# B&R Automation Studio project JOB_NUMBER (part 6)

#### SafetyUI.var - Local variables
```iecst
(********************************************************************
 * COPYRIGHT -- Bernecker + Rainer
 ********************************************************************
 * Program: SafetySample
 * File: SafetySample.var
 * Author: B&R
 ********************************************************************
 * Local variables of program SafetySample
 ********************************************************************)
VAR
	appcmd1 : DownloadCmdApplicationTypeV1; (*command structure for application download*)
	dataAcknMachineOptions : DownloadAcknMaOpTypeV1; (*data to acknowledge bit machine options*)
	datacmd1 : DownloadCmdMaOpTypeV1; (*command structure for machine options download*)
	datacmd2 : DownloadCmdExtMaOpTypeV1; (*command structure for extended machine options download*)
	dataMachineOptionsBitInput : ConfigurationBitOptionsTypeV1; (*data for bit machine options*)
	dataModuleFlagsInput : ConfigurationModuleFlagsTypeV1; (*data for module flags*)
	dialogApplication : BOOL; (*visualization dialog for application download*)
	dialogButtonLeft : BOOL; (*left button in visualization dialog*)
	dialogButtonRight : BOOL; (*right button in visualization dialog*)
	dialogData : BOOL; (*visualization dialog for machine options download*)
	dialogExtData : BOOL; (*visualization dialog for extended machine options download*)
	dialogRemoteCmd : BOOL; (*visualization dialog for remote control*)
	executeapp1 : BOOL; (*execute application download*)
	executedata1 : BOOL; (*execute machine options download*)
	executedata2 : BOOL; (*execute extended machine options download*)
	executeRemoteCmd : BOOL; (*execute remote control*)
	indexButtonLeft : UINT; (*index for button text*)
	indexButtonRight : UINT; (* index for button text*)
	indexCompareTextData : UINT; (*index for compare message machine options*)
	indexCompareTextExtData : UINT; (*index for compare message extended machine options*)
	indexFAILLed : UINT; (*index FAIL led*)
	indexFwAcknLed : UINT; (*index FW-ACKN led*)
	indexHeaderText : UINT; (*index dialog header text*)
	indexMessageText : UINT; (*index message text*)
	indexMxchgLed : UINT; (*index MXCHG led*)
	indexRELed : UINT; (*index R/E led*)
	Interface : STRING[80] := ''; (*interface information for SafeLOGIC*)
	Node : USINT; (*node information for SafeLOGIC*)
	pDeviceListOut : REFERENCE TO ARRAY[0..1] OF ConfigurationDeviceTypeV1; (*device list from FUB*)
	pMachineOptionsBitOut : REFERENCE TO ConfigurationBitOptionsTypeV1; (*bit machine options from FUB*)
	pModuleFlagsOut : REFERENCE TO ConfigurationModuleFlagsTypeV1; (*module flags form FUB*)
	readUDIDhighSL : EplSDORead; (*function block to read UDID high from device*)
	readUDIDhighSLX : AsIOAccRead; (*function block to read UDID high from device*)
	readUDIDlowSL : EplSDORead; (*function block to read UDID low from device*)
	readUDIDlowSLX : AsIOAccRead; (*function block to read UDID low from device*)
	remotecmd : RemoteControlCmdTypeV1; (*command structure for remote control*)
	safeDownloadApplication_0 : safeDownloadApplication; (*function block safeDownloadApplication*)
	safeDownloadData_0 : safeDownloadData; (*function block safeDownloadData*)
	safeDownloadData_1 : safeDownloadData; (*function block safeDownloadData*)
	safeRemoteControl_0 : safeRemoteControl; (*function block safeRemoteControl*)
	slxused : BOOL; (*SafeLOGIC-X is used*)
	Station : STRING[80] := 'IF6.ST1'; (*station information for SafeLOGIC-X*)
	statusAcknInfoData : UINT; (*acknowledge boxes for machine options*)
	statusAcknInfoExtData : UINT; (*acknowledge boxes for extended machine options*)
	statusButtonActiv : ARRAY[0..15] OF USINT; (*button activ*)
	statusButtonInactiv : ARRAY[0..15] OF USINT; (*button inactiv*)
	statusButtonUnlockApp : UINT; (*unlock buttons application*)
	statusButtonUnlockData : UINT; (*unlock buttons data*)
	statusButtonUnlockExtData : UINT; (*unlock buttons extended data*)
	statusDialog : UINT; (*dialog box*)
	statusSetPassword : UINT; (*visualization status to set password*)
	statusSLInformation : UINT; (*display information for SafeLOGIC*)
	stautsSLXInformation : UINT; (*display information for SafeLOGIC-X*)
	UDID_High : UINT; (*UDID_high for SafelOGIC*)
	UDID_Low : UDINT; (*UDID_low for SafeLOGIC*)
	visuAcknExtData : DownloadAcknExtMaOpTypeV1; (*acknowledge extended machine options*)
	visuAcknMachineOptions : ARRAY[0..511] OF BOOL; (*acknowledge machine options*)
	visuApplicationCRC : STRING[8]; (*CRC HEX string for visualization*)
	visuDeviceListInput : ARRAY[0..1] OF DownloadDeviceTypeV1; (*device list input*)
	visuDeviceListOutput : ARRAY[0..1] OF DownloadDeviceTypeV1; (*device list output*)
	visuDintInput : ConfigurationDintOptionsTypeV1; (*DINT channels input*)
	visuDintOutput : ConfigurationDintOptionsTypeV1; (*DINT channels output*)
	visuEnableDINTOptions : BOOL; (*enable DINT options*)
	visuEnableINTOptions : BOOL; (*enable INT options*)
	visuEnableMachineOptions : BOOL; (*enable BIT options*)
	visuEnableModuleFlags : BOOL; (*enable module flags*)
	visuEnableUDINTOptions : BOOL; (*enable UDINT options*)
	visuEnableUINTOptions : BOOL; (*enable UINT options*)
	visuIntInput : ConfigurationIntOptionsTypeV1; (*INT channels input*)
	visuIntOutput : ConfigurationIntOptionsTypeV1; (*INT channels output*)
	visuMachineOptionsBitInput : ARRAY[0..511] OF BOOL; (*BIT options input*)
	visuMachineOptionsBitOutput : ARRAY[0..511] OF BOOL; (*BIT options output*)
	visuModuleFlagsNotPresentInput : ARRAY[0..1023] OF BOOL; (*not present module flags input*)
	visuModuleFlagsNotPresentOutput : ARRAY[0..1023] OF BOOL; (*not present module flags output*)
	visuModuleFlagsOptionalInput : ARRAY[0..1023] OF BOOL; (*optional module flags input*)
	visuModuleFlagsOptionalOutput : ARRAY[0..1023] OF BOOL; (*optional module flags output*)
	visuModuleFlagsStartupInput : ARRAY[0..1023] OF BOOL; (*startup module flags input*)
	visuModuleFlagsStartupOutput : ARRAY[0..1023] OF BOOL; (*startup module flags output*)
	visuUDID_High : STRING[8]; (*UDID hex string for visualization*)
	visuUDID_Low : STRING[8]; (*UDID hex string for visualization*)
	visuUdintInput : ConfigurationUdintOptionsTypeV1; (*UDINT channels input*)
	visuUdintOutput : ConfigurationUdintOptionsTypeV1; (*UDINT channels output*)
	visuUintInput : ConfigurationUintOptionsTypeV1; (*UINT channels input*)
	visuUintOutput : ConfigurationUintOptionsTypeV1; (*UINT channels output*)
	visuUsedSLIDData : UINT; (*SafeLOGIC ID for data download*)
	visuUsedSLIDRemote : UINT; (*SafeLOGIC ID for remote control*)
	xcnt : UINT; (*counter variable*)
	strStatusID : STRING[10];
	strMXCHG_Led : STRING[10];
	strFWACKN_Led : STRING[10];
	strStatus : STRING[10];
	strRE_Led : STRING[10];
	strFAIL_Led : STRING[10];
	strMessageTest : STRING[10];
	bVisAppButtons : BOOL;
	bVisInterfaceNode : BOOL;
	bVisStation : BOOL;
	strDownloadStatus : STRING[10];
	strDataStatus : STRING[10];
	strSKFormatStyle : STRING[15];
	strSKXCHGtStyle : STRING[15];
	strScanStyle : STRING[15];
	strAck1Style : STRING[15];
	strAck2Style : STRING[15];
	strAck3Style : STRING[15];
	strAck4Style : STRING[15];
	strAckNStyle : STRING[15];
	strFWACKNStyle : STRING[15];
	strTestStyle : STRING[15];
	strClearStyle : STRING[15];
	safeLogicStatus : RemoteControlStatusTypeV1;
	visuEnableButtons : BOOL;
	safety : USINT;
	execute : BOOL;
	remoteControlcmd : REFERENCE TO RemoteControlCmdTypeV1;
	executeRemoteControl : BOOL;
	remoteCmdGetStatus : RemoteControlCmdTypeV1;
	ton_refreshStatus : TON_10ms;
	safePLC_Ok : BOOL;
	getNode : getNodeFromPV;
END_VAR
```

### Package Logical/COMMUNICATION - COMMUNICATION

### Communication.var
```iecst
(*Comm Config*)
VAR CONSTANT
  UDP_COMM_PORT : UINT := 4004;
  TCP_COMM_PORT : UINT := 12005;
END_VAR
(*Data sizes*)
VAR CONSTANT
  EVUE_COMM_BUFFER_SIZE : UINT := 16000; (*Size of data array for the memory map*)
  TCP_SEND_BUFFER_SIZE : UINT := 1000; (**Size of the send buffer for responses*)
  TCP_RECV_BUFFER_SIZE : UINT := 16000; (**Size of the recieve buffer*)
  UDP_SEND_PACKET_SIZE : UINT := 4000; (**Size of the packet to send*)
END_VAR
(***********UDP Comm Config************)
VAR CONSTANT
  LIVE_DATA_MAX_CONNECTIONS : USINT := 5; (**Maximum number of UDP Connections*)
  LIVE_DATA_MAX_POOL_SIZE : USINT := 10; (**Maximum number of data transmissions on 1 connection*)
END_VAR
(**)
(*DATA TYPE DEFINITIONS*)
VAR CONSTANT
  LIVE_DATA_TYPE_EVUE_UDP_COMM_1 : UINT := 1;
  LIVE_DATA_TYPE_EVUE_UDP_COMM_2 : UINT := 2;
  LIVE_DATA_TYPE_EVUE_UDP_COMM_3 : UINT := 3;
  LIVE_DATA_TYPE_EVUE_UDP_COMM_4 : UINT := 4;
  LIVE_DATA_TYPE_RAIL_MESSAGES : UINT := 1001;
END_VAR
(*DATA TYPE DEFINITIONS*)
VAR
        CommArray : ARRAY[0..EVUE_COMM_BUFFER_SIZE] OF UDINT; (**Global Array of pointers of comm vars*)
END_VAR
```

### Library Logical/COMMUNICATION/MbusTCP (ANSIC, version 1.39.0)
Depends on: astcp, asstring, standard, AsARCfg, sys_lib

### Program Logical/COMMUNICATION/ModSlave (IEC, version 2.00.1) - ModSlave

#### ModSlave.st - Init, cyclic, exit code
```iecst
(********************************************************************
  * COPYRIGHT --
  ********************************************************************
  * PROGRAM: ModSlave
  ********************************************************************
  * Implementation OF PROGRAM ModSlave
  ********************************************************************)

PROGRAM _INIT
  (* --------------------------------------------------------------------
    Reset FUNCTION blocks AND data structure on startup (SGC)
    --------------------------------------------------------------------- *)
  memset(ADR(ModbusTcpSlave), 0, SIZEOF(ModbusTcpSlave));
  memset(ADR(SlaveConfig), 0, SIZEOF(SlaveConfig));
  memset(ADR(logger), 0, SIZEOF(logger));

  (* --------------------------------------------------------------------
    Create default IO mapping FOR digital AND analog area
    --------------------------------------------------------------------- *)

  FOR idx:=0 TO SIZEOF(EVUE_MODBUS)/SIZEOF(EVUE_MODBUS[0])-1 DO
    SlaveConfig.p_holding_registers[idx] := ADR(EVUE_MODBUS[idx]);
  END_FOR;

  (* --------------------------------------------------------------------
    Configure FUNCTION block instance
    --------------------------------------------------------------------- *)
  ModbusTcpSlave.enable			:= 1; 					(* Enable function block *)
  ModbusTcpSlave.device			:= ADR('IF3');			(* Ethernet device string *)
  ModbusTcpSlave.p_cfg			:= ADR(SlaveConfig); 	(* IO configuration *)
  ModbusTcpSlave.master_timeout 	:= 5000; 			     	(* Disconnect master after x miliseconds when no request was sent, 0 = disabled *)

  (* The LOG information will show communication details. Enable for debugging,
  disable FOR production TO save system resources *)

  ModbusTcpSlave.log.data_lines 	:= 20; 					(* Number of logging lines *)
  ModbusTcpSlave.log.pData 		:= ADR(logger);			(* Pointer to logger string array *)
  mbSlaveStep := 1;
END_PROGRAM

PROGRAM _CYCLIC

  CASE mbSlaveStep OF
    0:
      (* --------------------------------------------------------------------
        Reset FUNCTION blocks AND data structure on startup (SGC)
        --------------------------------------------------------------------- *)
      memset(ADR(ModbusTcpSlave), 0, SIZEOF(ModbusTcpSlave));
      memset(ADR(SlaveConfig), 0, SIZEOF(SlaveConfig));
      memset(ADR(logger), 0, SIZEOF(logger));

      (* --------------------------------------------------------------------
        Configure FUNCTION block instance
        --------------------------------------------------------------------- *)
      ModbusTcpSlave.enable			:= 1; 					(* Enable function block *)
      ModbusTcpSlave.device			:= ADR('IF3');			(* Ethernet device string *)
      ModbusTcpSlave.p_cfg			:= ADR(SlaveConfig); 	(* IO configuration *)
      ModbusTcpSlave.master_timeout 	:= 5000; 			     	(* Disconnect master after x miliseconds when no request was sent, 0 = disabled *)

      // Go to mbSlaveStep 1
      mbSlaveStep := 1;

    1:
      // Call MbSlave FUB
      ModbusTcpSlave();
  END_CASE

  (* --------------------------------------------------------------------
    Reset last error information
    --------------------------------------------------------------------- *)
  IF(reset_error) THEN
    memset(ADR(ModbusTcpSlave.last_error), 0, 2);
    reset_error := 0;
  END_IF
END_PROGRAM
```

### Program Logical/COMMUNICATION/udpComm (IEC, version 2.00.1) - udpComm

#### Main.st - Init, cyclic, exit code
```iecst
(*
  ----------------------------------------------------------------------------------------------------------------------------------------
  --LIVE DATA TASK--
  UDP MAX FRAME SIZE IS 65507 Bytes
  -----------------------------------------------------------------------------------------------------------------------------------------
  *)
  //V1.00.1 -- 06/09/2019 -- First Version
  //V1.00.2 -- 05/01/2020 -- Clean up basic version + Add dynamic start up for ABB drive data
  //V2.00.1 -- 11/03/2020 -- Add Structures to replace TCP/IP Driver
  PROGRAM _INIT
  //Configure a static connection (Testing)
  LiveDataConnection[1].Config.ServerIP 		:= eVueServerIP;
  LiveDataConnection[1].Config.ServerPort		:= UDP_COMM_PORT;
  LiveDataConnection[1].Config.Type 			:= LIVE_DATA_CONFIG_STATIC;
  //Create a fix request pool for test
  LiveDataConnection[1].RequestPool.PoolList[1] 	:= LIVE_DATA_TYPE_EVUE_UDP_COMM_1;
  LiveDataConnection[1].RequestPool.PoolList[2] 	:= LIVE_DATA_TYPE_EVUE_UDP_COMM_2;
  LiveDataConnection[1].RequestPool.PoolList[3] 	:= LIVE_DATA_TYPE_EVUE_UDP_COMM_3;
  LiveDataConnection[1].RequestPool.PoolList[4] 	:= LIVE_DATA_TYPE_EVUE_UDP_COMM_4;
  LiveDataConnection[1].RequestPool.PoolList[5] 	:= LIVE_DATA_TYPE_RAIL_MESSAGES;
  LiveDataConnection[1].RequestPool.PoolListSize 	:= 5;
  _initialiseComms;
  END_PROGRAM

  PROGRAM _CYCLIC

    IF EDGEPOS(udpIdent_Error) THEN
      udpCloseAllIdent := 0;
      n := 0;
    END_IF;
    IF udpIdent_Error THEN // We have too many ports open -- temp stop all clients and close all udp connections.

      CASE udpCloseAllIdent OF

      0://Get list off all open idents
        ioctl ACCESS ADR(udpIoctl_Error);
        ioctl.enable := 1;
        ioctl.ident := udpINVALID_IDENT;
        ioctl.ioctl := udpID_LIST_GET;
        ioctl.pData := ADR(identInfo.IdentsList[0]);
        ioctl.datalen := SIZEOF(identInfo.IdentsList);
        ioctl();
        IF (ioctl.status = ERR_OK) THEN
          udpCloseAllIdent := 1;
        ELSIF (ioctl.status <> ERR_FUB_BUSY) THEN

        END_IF;

      1://Close all open connections

        close ACCESS ADR(udpClose_Error);
        close.enable := (identInfo.IdentsList[n] > 0);
        close.ident := identInfo.IdentsList[n];
        close();
        IF (close.status = ERR_OK) OR ((close.status <> ERR_FUB_BUSY) AND (close.status <> ERR_FUB_ENABLE_FALSE)) THEN
          identInfo.IdentsList[n] := 0;
          IF (n < 199) THEN
            n := n + 1;
          ELSE
            udpCloseAllIdent := 2;
          END_IF;
        ELSIF (identInfo.IdentsList[n] = 0) THEN
          udpCloseAllIdent := 2;
        END_IF;

      2:// Reinint all connections
        FOR n := 1 TO LIVE_DATA_MAX_CONNECTIONS DO
          connection ACCESS ADR(LiveDataConnection[n]);
          connection.State := LIVE_DATA_INIT;
        END_FOR;
        udpIdent_Error := 0;
        udpCloseAllIdent := 0;
      END_CASE;

    ELSE //Run
      FOR n := 1 TO LIVE_DATA_MAX_CONNECTIONS DO
        connection ACCESS ADR(LiveDataConnection[n]);
        CASE connection.State  OF
          LIVE_DATA_INIT: //Every connection must be initialised with server IP and Port. This can be static or dynamic via http GET.
            CASE connection.Config.Type OF
              LIVE_DATA_CONFIG_STATIC:
                //Check the IP is valid
                IF connection.Config.ServerIP <> '' THEN //Don;t check Port as this could be 0
                  connection.State := LIVE_DATA_WAIT;
                END_IF;
              LIVE_DATA_CONFIG_DYNAMIC_CLIENT:
                //Http request to load the Server details + current request pool
              LIVE_DATA_CONFIG_DYNAMIC_SERVER;
                //Wait for a request on the http server to start a connection.
            END_CASE;

          LIVE_DATA_WAIT:
            _AddRemoveFromPool;
            //Wait for the Request pool to be greater than 0
            IF (connection.RequestPool.PoolListSize > 0) THEN
              connection.State := LIVE_DATA_OPEN_CONNECTION;
            END_IF;

          LIVE_DATA_OPEN_CONNECTION:
            //Open connection to serverr
            open ACCESS ADR(connection.Functions.Open);
            open.enable 	:= 1;
            open.options	:= 0;
            open.pIfAddr 	:= 0;//
            open.port		:= 0;//
            open();
            IF (open.status = ERR_OK) THEN
              connection.State := LIVE_DATA_SETUP_CONNECTION_TOS;
            ELSIF (open.status <> ERR_FUB_BUSY) THEN
              connection.Error := open.status;
              connection.State := LIVE_DATA_ERROR; // Go directly to error as the connection has failed
            END_IF;

          LIVE_DATA_SETUP_CONNECTION_TOS://Configure the UDP
            //We must set
            //1) Type of service 	-- udpIP_TOS_SET -- udpIP_TOS_RELIABILITY
            //2) Time to live 		--
            //Optional Send Buffer	-- udpSO_SNDBUF_SET

            //				udpIP_TOS_LOWDELAY			16
            //				udpIP_TOS_THROUGHPUT		8
            //				udpIP_TOS_RELIABILITY		4
            //				udpIP_TOS_MINCOST			2

            ioctl ACCESS ADR(connection.Functions.Ioctl);
            ioctl.enable := 1;
            ioctl.ident := connection.Functions.Open.ident;
            ioctl.ioctl := udpIP_TOS_SET;
            ioctl.pData := ADR(connection.Config.TOS);
            ioctl.datalen := 4;
            ioctl();
            IF (ioctl.status = ERR_OK) THEN
              connection.State := LIVE_DATA_SETUP_CONNECTION_TTL;
            ELSIF (ioctl.status <> ERR_FUB_BUSY) THEN
              connection.Error := ioctl.status;
              connection.State := LIVE_DATA_CLOSE_CONNECTION;
            END_IF;

          LIVE_DATA_SETUP_CONNECTION_TTL: //Time to LIVE in seconds -- MAX 255

            ioctl ACCESS ADR(connection.Functions.Ioctl);
            ioctl.enable := 1;
            ioctl.ident := connection.Functions.Open.ident;
            ioctl.ioctl := udpIP_TTL_SET;
            ioctl.pData := ADR(connection.Config.TTL);
            ioctl.datalen := 4;
            ioctl();
            IF (ioctl.status = ERR_OK) THEN
              connection.State := LIVE_DATA_CONNECT;
            ELSIF (ioctl.status <> ERR_FUB_BUSY) THEN
              connection.Error := ioctl.status;
              connection.State := LIVE_DATA_CLOSE_CONNECTION;
            END_IF;

          LIVE_DATA_CONNECT: // Connect to a specific Device (this is optional but improves performance)
            connect	ACCESS ADR(connection.Functions.Connect);
            connect.enable 	:= 1;
            connect.ident 	:= connection.Functions.Open.ident;
            connect.pHost	:= ADR(connection.Config.ServerIP);
            connect.port 	:= connection.Config.ServerPort;
            connect();
            IF (connect.status = ERR_OK) THEN
              IF getIdentInfo THEN
                connection.State := LIVE_DATA_GET_IDENT_LIST;
              ELSE
                connection.State := LIVE_DATA_BUILD_DATA;
              END_IF;
            ELSIF (connect.status <> ERR_FUB_BUSY) THEN
              connection.Error := connect.status;
              connection.State := LIVE_DATA_DISCONNECT;
            END_IF;
          LIVE_DATA_BUILD_DATA:
            //Build data-- Build a header and data combined.
            //Byte 1 		-- Request Type USINT
            //Byte 2 & 3	-- Header Size(Bytes) UINT
            //Byte 4,5,6,7	-- CheckSum		UDINT
            //Byte xxx		-- HEADER INFO -- BESPOKE TO Request Type
            //DATA--
            IF (connection.RequestPool.Pointer > 0) THEN
              CASE connection.RequestPool.PoolList[connection.RequestPool.Pointer] OF

                LIVE_DATA_TYPE_EVUE_UDP_COMM_1..LIVE_DATA_TYPE_EVUE_UDP_COMM_4:
                  //Built the packet
                  udpComm[0] := connection.RequestPool.Pointer;
                  FOR n := 1 TO UDP_SEND_PACKET_SIZE DO
                    pointer :=  n + (UDP_SEND_PACKET_SIZE * (udpComm[0] - 1));
                    IF (CommArray[pointer] <> 0) AND (pointer <= EVUE_COMM_BUFFER_SIZE) THEN
                      brsmemcpy(ADR(udpComm[n]),CommArray[pointer],2);
                    ELSE
                      udpComm[n] := 0;
                    END_IF;
                  END_FOR;
                  pData := ADR(udpComm);
                  length := SIZEOF(udpComm);
                  connection.State := LIVE_DATA_SEND_DATA;

                LIVE_DATA_TYPE_RAIL_MESSAGES:// Rail messages
                  messages[0] := LIVE_DATA_TYPE_RAIL_MESSAGES;
                  FOR n := 1 TO RAIL_COUNT DO
                    messages[n] := RailComm[n].Messages.Write;
                  END_FOR;
                  pData := ADR(messages);
                  length := SIZEOF(messages);
                  connection.State := LIVE_DATA_SEND_DATA;

                ELSE
                  //Invalid type- Check the pool again
                  connection.State := LIVE_DATA_CHECK_REQUESTPOOL;
              END_CASE;
            ELSE
              connection.State := LIVE_DATA_CHECK_REQUESTPOOL;
            END_IF;

          LIVE_DATA_SEND_DATA:
            send ACCESS ADR(connection.Functions.Send);
            send.enable 	:= 1;
            send.ident 		:= connection.Functions.Open.ident;
            send.flags 		:= udpMSG_DONTROUTE;// Do not send via the gateway- Route Directly to Server
            send.pData 		:= pData;
            send.datalen	:= length;
            send();
            IF (send.status = ERR_OK) THEN
              connection.State := LIVE_DATA_CHECK_REQUESTPOOL;
            ELSIF send.status = udpERR_CONNREFUSED THEN // Server is not there, disconnect and start again
              connection.State := LIVE_DATA_DISCONNECT;
            ELSIF (send.status <> ERR_FUB_BUSY) THEN
              connection.Error := send.status;
              connection.State := LIVE_DATA_DISCONNECT;
            END_IF;

            //send.pHost || THESE ARE IGNORED BECAUSE WE ARE MAKING A DIRECT CONNECTION USING THE CONNECT FUB||
            //send.port

          LIVE_DATA_CHECK_REQUESTPOOL:
            //Check that the request pool hasn;t changed- Shuffle to the next Requested packet.
            _AddRemoveFromPool;
            //IF the pool is empty close the connection and wait
            IF (connection.RequestPool.Pointer = 0) AND (connection.RequestPool.PoolListSize > 0) THEN
              connection.RequestPool.Pointer := 1;
            ELSIF (connection.RequestPool.Pointer = connection.RequestPool.PoolListSize) THEN
              connection.RequestPool.Pointer := 1;
            ELSIF (connection.RequestPool.Pointer < connection.RequestPool.PoolListSize) THEN
              connection.RequestPool.Pointer := connection.RequestPool.Pointer + 1;
            ELSIF (connection.RequestPool.Pointer > connection.RequestPool.PoolListSize) AND (connection.RequestPool.PoolListSize > 0) THEN
              connection.RequestPool.Pointer := 1;
            END_IF;

            validConnection := (connection.Config.ServerIP <> '');
            IF (connection.RequestPool.PoolListSize = 0) OR NOT validConnection THEN
              connection.State := LIVE_DATA_DISCONNECT;
            ELSE
              connection.State := LIVE_DATA_BUILD_DATA;
            END_IF;

          LIVE_DATA_DISCONNECT:
            disconnect ACCESS ADR(connection.Functions.Disconnect);
            disconnect.enable := 1;
            disconnect.ident := connection.Functions.Open.ident;
            disconnect();
            IF (disconnect.status = ERR_OK) THEN
              connection.State := LIVE_DATA_CLOSE_CONNECTION;
            ELSIF (disconnect.status <> ERR_FUB_BUSY) THEN
              connection.Error := disconnect.status;
              connection.State := LIVE_DATA_CLOSE_CONNECTION;
            END_IF;

          LIVE_DATA_CLOSE_CONNECTION:
            close ACCESS ADR(connection.Functions.Close);
            close.enable := 1;
            close.ident := connection.Functions.Open.ident;
            close();
            IF (close.status = ERR_OK) THEN
              IF (connection.Error > 0) THEN
                connection.State := LIVE_DATA_ERROR;
              ELSE
                connection.State := LIVE_DATA_INIT;
              END_IF;
              IF (connection.Config.Type <> LIVE_DATA_CONFIG_STATIC) THEN
                connection.RequestPool 			:= CLEAR_REQUEST_POOL;
                connection.Config.ServerIP 		:= '';
                connection.Config.ServerPort 	:= 0;
              END_IF;

            ELSIF (close.status <> ERR_FUB_BUSY) THEN
              connection.Error := close.status ;
              connection.State := LIVE_DATA_ERROR;
            END_IF;

          LIVE_DATA_ERROR:
            IF (connection.Error = udpERR_NOMORE_IDENTS) THEN
              // All Idents are used we have to close them manually.
              udpIdent_Error := 1;
            ELSE
              errorCount := errorCount + 1;
              connection.Error := 0;
              connection.State := LIVE_DATA_INIT;
            END_IF;

          LIVE_DATA_GET_IDENT_LIST:
            ioctl ACCESS ADR(connection.Functions.Ioctl);
            ioctl.enable := 1;
            ioctl.ident := udpINVALID_IDENT;
            ioctl.ioctl := udpID_LIST_GET;
            ioctl.pData := ADR(identInfo.IdentsList[0]);
            ioctl.datalen := SIZEOF(identInfo.IdentsList);
            ioctl();
            IF (ioctl.status = ERR_OK) THEN
              connection.State := LIVE_DATA_GET_IDENT_MAX;
            ELSIF (ioctl.status <> ERR_FUB_BUSY) THEN

            END_IF;

          LIVE_DATA_GET_IDENT_MAX:
            ioctl ACCESS ADR(connection.Functions.Ioctl);
            ioctl.enable := 1;
            ioctl.ident := udpINVALID_IDENT;
            ioctl.ioctl := udpID_MAX_GET;
            ioctl.pData := ADR(identInfo.MaxIdents);
            ioctl.datalen := 4;
            ioctl();
            IF (ioctl.status = ERR_OK) THEN
              connection.State := LIVE_DATA_BUILD_DATA;
            ELSIF (ioctl.status <> ERR_FUB_BUSY) THEN

            END_IF;

        END_CASE;

      END_FOR;
    END_IF;

  END_PROGRAM

  PROGRAM _EXIT
    // DO we have to close the connections on EXIT -- Perhaps when a transfer happens!!

  END_PROGRAM
```

#### _AddRemoveFromPool.st
```iecst
ACTION _AddRemoveFromPool:
IF (connection.RequestPool.AddToPool > 0) THEN
  //Check the requested frame is not already in the list
  FOR i := 1 TO LIVE_DATA_MAX_POOL_SIZE DO
    IF (connection.RequestPool.PoolList[i] = connection.RequestPool.AddToPool) THEN
      connection.RequestPool.AddToPool := 0;
      EXIT;
    ELSIF (connection.RequestPool.PoolList[i] = 0) THEN
      EXIT;
    END_IF;
  END_FOR;

  IF (connection.RequestPool.AddToPool > 0) THEN //Check we haven't already found the request in the pool
    IF (connection.RequestPool.PoolListSize < LIVE_DATA_MAX_POOL_SIZE) THEN //Keep in range
      connection.RequestPool.PoolListSize := connection.RequestPool.PoolListSize + 1;
      connection.RequestPool.PoolList[connection.RequestPool.PoolListSize] := connection.RequestPool.AddToPool;
      connection.RequestPool.AddToPool := 0;
    END_IF;
  END_IF;
END_IF;
IF (connection.RequestPool.RemoveFromPool > 0) THEN
  //Find the pool in the array-- Remove it then shuffle the list.
  FOR i := 1 TO LIVE_DATA_MAX_POOL_SIZE DO
    IF (connection.RequestPool.PoolList[i] = connection.RequestPool.RemoveFromPool) THEN
      //Shuffle the list
      brsmemmove(ADR(connection.RequestPool.PoolList[i]),ADR(connection.RequestPool.PoolList[i + 1]),((LIVE_DATA_MAX_POOL_SIZE - i)*2));
      //connection.RequestPool.PoolList[LIVE_DATA_MAX_POOL_SIZE] := 0;
      connection.RequestPool.PoolListSize := connection.RequestPool.PoolListSize - 1;
      IF (connection.RequestPool.PoolListSize > LIVE_DATA_MAX_POOL_SIZE) THEN
        connection.RequestPool.PoolListSize := 0;
      END_IF;
      EXIT;
    ELSIF (connection.RequestPool.PoolList[i] = 0) THEN
      EXIT; //Not found
    END_IF;
  END_FOR;
  connection.RequestPool.RemoveFromPool := 0;
END_IF;
END_ACTION
```

#### _initialiseComms.st
```iecst
// Initialise the Comm registers.
ACTION _initialiseComms:
  //Generated Init Code.
  FOR n := 0 TO EVUE_COMM_BUFFER_SIZE DO
    CommArray[n] := 0;
  END_FOR;

END_ACTION
```

#### Types.typ - Local data types
```iecst
TYPE
  identInfo_typ : 	STRUCT
    MaxIdents : UDINT;
    IdentsList : ARRAY[0..199]OF UDINT;
  END_STRUCT;
END_TYPE
```

#### Variables.var - Local variables
```iecst
VAR CONSTANT
  CLEAR_REQUEST_POOL : LiveData_RequestPool_typ := (AddToPool:=0,RemoveFromPool:=0,PoolListSize:=0,Pointer:=0);
END_VAR
VAR
  n : UINT;
  pointer : UDINT;
  connection : REFERENCE TO LiveDataConnection_typ;
  LiveDataConnection : ARRAY[1..LIVE_DATA_MAX_CONNECTIONS] OF LiveDataConnection_typ;
  udpComm : ARRAY[0..UDP_SEND_PACKET_SIZE] OF UINT;
  open : REFERENCE TO UdpOpen;
  ioctl : REFERENCE TO UdpIoctl;
  connect : REFERENCE TO UdpConnect;
  send : REFERENCE TO UdpSend;
  pData : UDINT;
  length : UDINT;
  disconnect : REFERENCE TO UdpDisconnect;
  close : REFERENCE TO UdpClose;
  errorCount : UDINT;
  validConnection : BOOL;
  i : USINT;
  identInfo : identInfo_typ;
  getIdentInfo : BOOL;
  udpIdent_Error : BOOL;
  udpIoctl_Error : UdpIoctl;
  udpCloseAllIdent : USINT;
  udpClose_Error : UdpClose;
  data : ARRAY[0..65534] OF SINT; (**Max data frame that can be sent by UDP*)
  messages : ARRAY[0..RAIL_COUNT] OF UINT;
END_VAR
```

### Program Logical/COMMUNICATION/tcpComm (IEC, version 1.00.1) - tcpComm

#### Main.st - Init, cyclic, exit code
```iecst
//V1.00 	- First Version
//V1.00.1 	- ADD Evue modbus decode function.
PROGRAM _INIT
  _initialiseComms;
	listenPort 	:= TCP_COMM_PORT;
	socketState := TCP_SOCKET_OPEN;
END_PROGRAM
PROGRAM _CYCLIC

	CASE socketState OF
		TCP_SOCKET_OPEN:
			tcpOpen.enable := 1;
			tcpOpen.options := tcpOPT_REUSEADDR;
			tcpOpen.pIfAddr := 0; //Listen for any connection
			tcpOpen.port := listenPort;
			tcpOpen();
			IF (tcpOpen.status = ERR_OK) THEN
				socketState := TCP_SOCKET_LISTEN;
			ELSIF tcpOpen.status <> ERR_FUB_BUSY THEN
				socketState := TCP_SOCKET_GET_CONNECTION_LIST; // Close all connections if we have any socket errors
			END_IF;

		TCP_SOCKET_LISTEN:
			tcpServer.enable := (tcpOpen.ident > 0);
			tcpServer.ident := tcpOpen.ident;
			tcpServer.backlog := MAX_TCP_CONNECTIONS; //Only this many connections
			tcpServer.pIpAddr := ADR(ipAddress);
			tcpServer();
			IF tcpServer.status = ERR_OK THEN
				connectCount := connectCount + 1; // DEBUG INFO ONLY
				FOR n := 0 TO MAX_TCP_CONNECTIONS DO // Find an available server
					IF (server[n].State = TCP_SERVER_IDLE) AND (server[n].Ident = 0) THEN
						server[n].Ident			:= tcpServer.identclnt;
						server[n].ResponsePort 	:= tcpServer.portclnt;
						server[n].IpAddress 	:= ipAddress;
						EXIT;
					END_IF;
				END_FOR;
			ELSIF tcpServer.status <> ERR_FUB_BUSY THEN
				socketState := TCP_SOCKET_GET_CONNECTION_LIST; // Close all connections if we have any socket errors.
			END_IF;

		TCP_SOCKET_GET_CONNECTION_LIST:
			tcp_Ioctl.enable := 1;
			tcp_Ioctl.ident := tcpINVALID_IDENT;
			tcp_Ioctl.ioctl := tcpID_LIST_GET;
			tcp_Ioctl.pData := ADR(usedIdentList[0]);
			tcp_Ioctl.datalen := SIZEOF(usedIdentList);
			tcp_Ioctl();
			IF (tcp_Ioctl.status = ERR_OK) THEN
				x := 0;
				socketState := TCP_SOCKET_CLOSE_ALL_CONNECTIONS;
			ELSIF (tcp_Ioctl.status <> ERR_FUB_BUSY) THEN
				socketState := TCP_SOCKET_OPEN;//TCP_SOCKET_ERROR;
			END_IF;

		TCP_SOCKET_CLOSE_ALL_CONNECTIONS:

			//WHILE (usedIdentList[n] <> 0) DO  // Remove the While loop- PLC can;t cope in 10ms
			socketClose.enable := (usedIdentList[x] > 0);
			socketClose.ident := usedIdentList[x];
			socketClose.how  := 0;// (tcpSHUT_RD OR tcpSHUT_WR); // Bitwise- set both flags.
			socketClose();
			IF (socketClose.status = ERR_OK) THEN
				usedIdentList[x] := 0;
				IF x < 254 THEN x:= x + 1; END_IF;
			ELSIF (socketClose.status <> ERR_FUB_BUSY) THEN
				usedIdentList[x] := 0;
				IF x < 254 THEN x:= x + 1; END_IF;
			END_IF;
			//END_WHILE;
			IF (usedIdentList[x] = 0) THEN
				socketState := TCP_SOCKET_OPEN;
			END_IF;

		TCP_SOCKET_ERROR:

	END_CASE

	//Handle each server state..
	FOR n := 0 TO MAX_TCP_CONNECTIONS DO

		IF (socketState = TCP_SOCKET_LISTEN) THEN

			//Set up the references
			_references;

			//Close the connection after 60'
			ton_NoData.IN := (state = TCP_SERVER_RECV);
			ton_NoData.PT := T#60s;
			ton_NoData();

			CASE state OF

				TCP_SERVER_IDLE:
					IF ident > 0 THEN
						state := TCP_SERVER_RECV;
					END_IF;

				TCP_SERVER_RECV:
					tcpRecv.enable := (ident > 0);
					tcpRecv.ident := ident;
					tcpRecv.pData := ADR(server[n].RecieveData[0]);
					tcpRecv.datamax := SIZEOF(server[n].RecieveData);
					tcpRecv.flags := 0;
					tcpRecv();
					IF tcpRecv.status = ERR_OK AND (tcpRecv.recvlen > 0)  THEN
//						Open the packet TO decide how TO deocde it
// 						FIRST WORD MUSE BE PACKET TYPE
						CASE server[n].RecieveData[0] OF
							1: // eVue Modbus replacement.
								_decodeModbus;
							100://ECHO
								IF (tcpRecv.recvlen <= TCP_SEND_BUFFER_SIZE) THEN
									memcpy(ADR(server[n].SendData[0]),ADR(server[n].RecieveData[0]),tcpRecv.recvlen);
									sendSize[n] := tcpRecv.recvlen;
								ELSE // Only respond as much as we can.
									memcpy(ADR(server[n].SendData[0]),ADR(server[n].RecieveData[0]),TCP_SEND_BUFFER_SIZE);
									sendSize[n] := TCP_SEND_BUFFER_SIZE;
								END_IF;
								state := TCP_SERVER_SEND;
              1001: // Message Acknowledge
                _messageAcknowledge;
              ELSE // Fail to DECODE -- Send fail message.
								brsstrcpy(ADR(server[n].SendData[0]),ADR(TCP_FAIL_DECODE));
								sendSize[n] := LEN(TCP_FAIL_DECODE);
								state := TCP_SERVER_SEND;
						END_CASE;
					ELSIF (tcpRecv.status = tcpERR_NOT_CONNECTED) THEN
						state := TCP_SERVER_CLOSE;
					ELSIF (tcpRecv.status = tcpERR_NO_DATA) THEN
						//state := TCP_SERVER_SEND;
					ELSIF(tcpRecv.status <> ERR_FUB_BUSY) THEN
						state := TCP_SERVER_CLOSE;
					ELSIF ton_NoData.Q THEN
						state := TCP_SERVER_CLOSE;
					ELSIF (ident = 0) THEN
						server[n] := SERVER_IDLE;
					END_IF;

				TCP_SERVER_SEND:
					tcpSend.enable := (ident > 0);
					tcpSend.ident := ident;
					tcpSend.pData := ADR(server[n].SendData[0]);
					tcpSend.datalen := sendSize[n];
					tcpSend.flags := 0;
					tcpSend();
					IF tcpSend.status = ERR_OK THEN
						state := TCP_SERVER_RECV;
					ELSIF (tcpSend.status <> ERR_FUB_BUSY) THEN
						state := TCP_SERVER_CLOSE;
					ELSIF (ident = 0) THEN
						server[n] := SERVER_IDLE;
					END_IF;

				TCP_SERVER_CLOSE:
					tcpClose.enable := (ident > 0);
					tcpClose.how	:= 0;
					tcpClose.ident	:= ident;
					tcpClose();
					IF tcpClose.status = ERR_OK THEN
						ident := 0;
						server[n] := SERVER_IDLE;
					ELSIF tcpClose.status <> ERR_FUB_BUSY THEN
						ident := 0;
						server[n] := SERVER_IDLE;
					END_IF;

			END_CASE;

			IF EDGEPOS(state = TCP_SERVER_RECV) THEN
				memset(ADR(server[n].SendData[0]),0,SIZEOF(server[n].SendData));
				memset(ADR(server[n].RecieveData[0]),0,SIZEOF(server[n].RecieveData));
			END_IF;
		ELSE
			server[n] := SERVER_IDLE;
		END_IF;
	END_FOR;

END_PROGRAM
PROGRAM _EXIT

END_PROGRAM
```
